# EPICS autosave request: peakAnalyserApp/Db/peakAnalyser_settings.req
file "ADBase_settings.req", P=$(P), R=$(R)
#$(P)$(R)LENS_MODE
#$(P)$(R)DETECTOR_MODE
#$(P)$(R)PASS_ENERGY
#$(P)$(R)ACQ_MODE
#$(P)$(R)ENERGY_MODE
#$(P)$(R)EXCITATION_ENERGY
$(P)$(R)LOW_ENERGY
$(P)$(R)HIGH_ENERGY
$(P)$(R)CENTRE_ENERGY
$(P)$(R)STEP_SIZE
$(P)$(R)LOW_THETA_Y
$(P)$(R)HIGH_THETA_Y
$(P)$(R)CENTRE_THETA_Y
$(P)$(R)THETA_Y_STEP_SIZE
$(P)$(R)CENTRE_SLICE
$(P)$(R)CHANNELS
$(P)$(R)SLICES
